FUNCTION_BLOCK FB_MotionAxisDS402NCSync EXTENDS FB_MotionAxisDS402NC
VAR_INPUT
END_VAR
VAR_OUTPUT
END_VAR
VAR
    iMotionAxisShareData : I_MotionAxisShareData;
END_VAR

// read  shared data

// call super class body
SUPER^();

// Write shared data

(*FB_Init is always available implicitly and it is used primarily for initialization.
The return value is not evaluated. For a specific influence, you can also declare the
methods explicitly and provide additional code there with the standard initialization
code. You can evaluate the return value.*)
METHOD FB_Init : BOOL
VAR_INPUT
    (* TRUE: the retain variables are initialized (reset warm / reset cold)*)
    bInitRetains	: BOOL;
    (* TRUE: the instance will be copied to the copy code afterward (online change)*)
    bInCopyCode	: BOOL;
    AxisRef	: REFERENCE TO AXIS_REF;
    iPersistentDataStorage	: I_PersistentDataStorage;
    iMotionLogger	: I_MotionLogger;
    iDS402DriveCommon 	: I_DS402DriveCommon;
    ModeOfOperation : E_DS402OpMode;
    iMotionAxisShareData : I_MotionAxisShareData;

END_VAR
THIS^.iMotionAxisShareData :=  iMotionAxisShareData;
END_METHOD

END_FUNCTION_BLOCK

(* stored: Version 1.1.0.1
   POU FB_MotionAxisDS402NCSync: Id {0e4f30c7-9701-46fd-b9a3-891c9877e9a0}, SpecialFunc None
   Method FB_Init: Id {1dac3e04-3581-442d-91f0-9c2dc1b453ee} *)
